// SIMATIC S7-200 project (STEP 7-Micro/WIN), CPU 224 REL 02.01

SYMBOL_TABLE USER1
start            M0.0     // khoi dong
stopp            M0.1     // dung dong co
CBT              M0.2     // cam bien quay phai
CBP              M0.3     // cam bien quay trai
QT               M0.4     // QUAY TRAI
QP               M0.5     // QUAY PHAI
END_SYMBOL_TABLE

ORGANIZATION_BLOCK MAIN:OB1
TITLE=PROGRAM COMMENTS
BEGIN
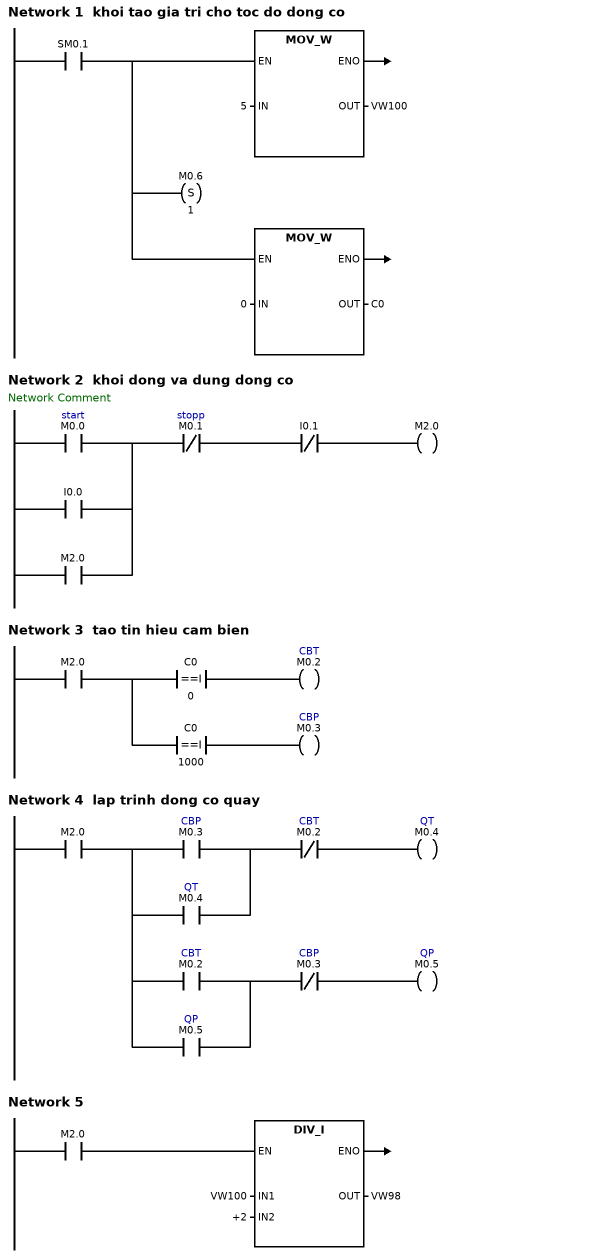
Network 1 // khoi tao gia tri cho toc do dong co
LD     SM0.1
MOVW   5, VW100
S      M0.6, 1
MOVW   0, C0
Network 2 // khoi dong va dung dong co
// Network Comment
LD     start:M0.0
O      I0.0
O      M2.0
AN     stopp:M0.1
AN     I0.1
=      M2.0
Network 3 // tao tin hieu cam bien
LD     M2.0
LPS
AW=    C0, 0
=      CBT:M0.2
LPP
AW=    C0, 1000
=      CBP:M0.3
Network 4 // lap trinh dong co quay
LD     M2.0
LPS
LD     CBP:M0.3
O      QT:M0.4
ALD
AN     CBT:M0.2
=      QT:M0.4
LPP
LD     CBT:M0.2
O      QP:M0.5
ALD
AN     CBP:M0.3
=      QP:M0.5
Network 5
LD     M2.0
MOVW   VW100, VW98
/I     +2, VW98
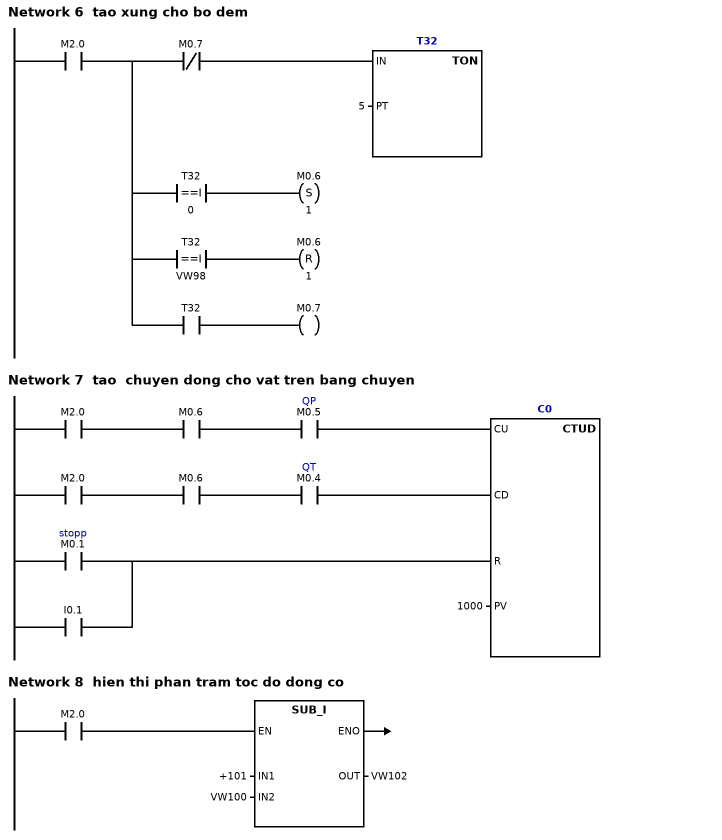
Network 6 // tao xung cho bo dem
LD     M2.0
LPS
AN     M0.7
TON    T32, 5
LRD
AW=    T32, 0
S      M0.6, 1
LRD
AW=    T32, VW98
R      M0.6, 1
LPP
A      T32
=      M0.7
Network 7 // tao  chuyen dong cho vat tren bang chuyen
LD     M2.0
A      M0.6
A      QP:M0.5
LD     M2.0
A      M0.6
A      QT:M0.4
LD     stopp:M0.1
O      I0.1
CTUD   C0, 1000
Network 8 // hien thi phan tram toc do dong co
LD     M2.0
MOVW   +101, VW102
-I     VW100, VW102
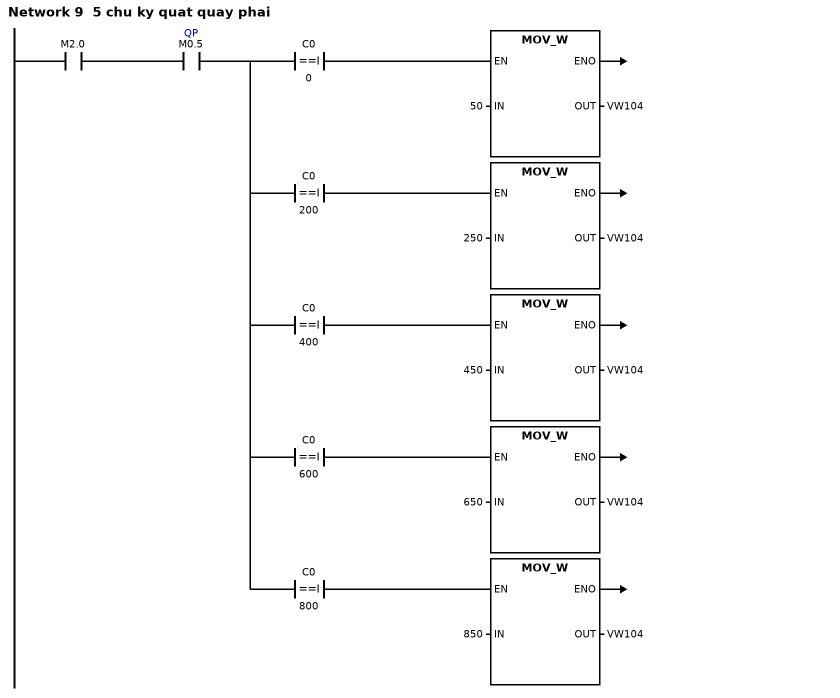
Network 9 // 5 chu ky quat quay phai
LD     M2.0
A      QP:M0.5
LPS
AW=    C0, 0
MOVW   50, VW104
LRD
AW=    C0, 200
MOVW   250, VW104
LRD
AW=    C0, 400
MOVW   450, VW104
LRD
AW=    C0, 600
MOVW   650, VW104
LPP
AW=    C0, 800
MOVW   850, VW104
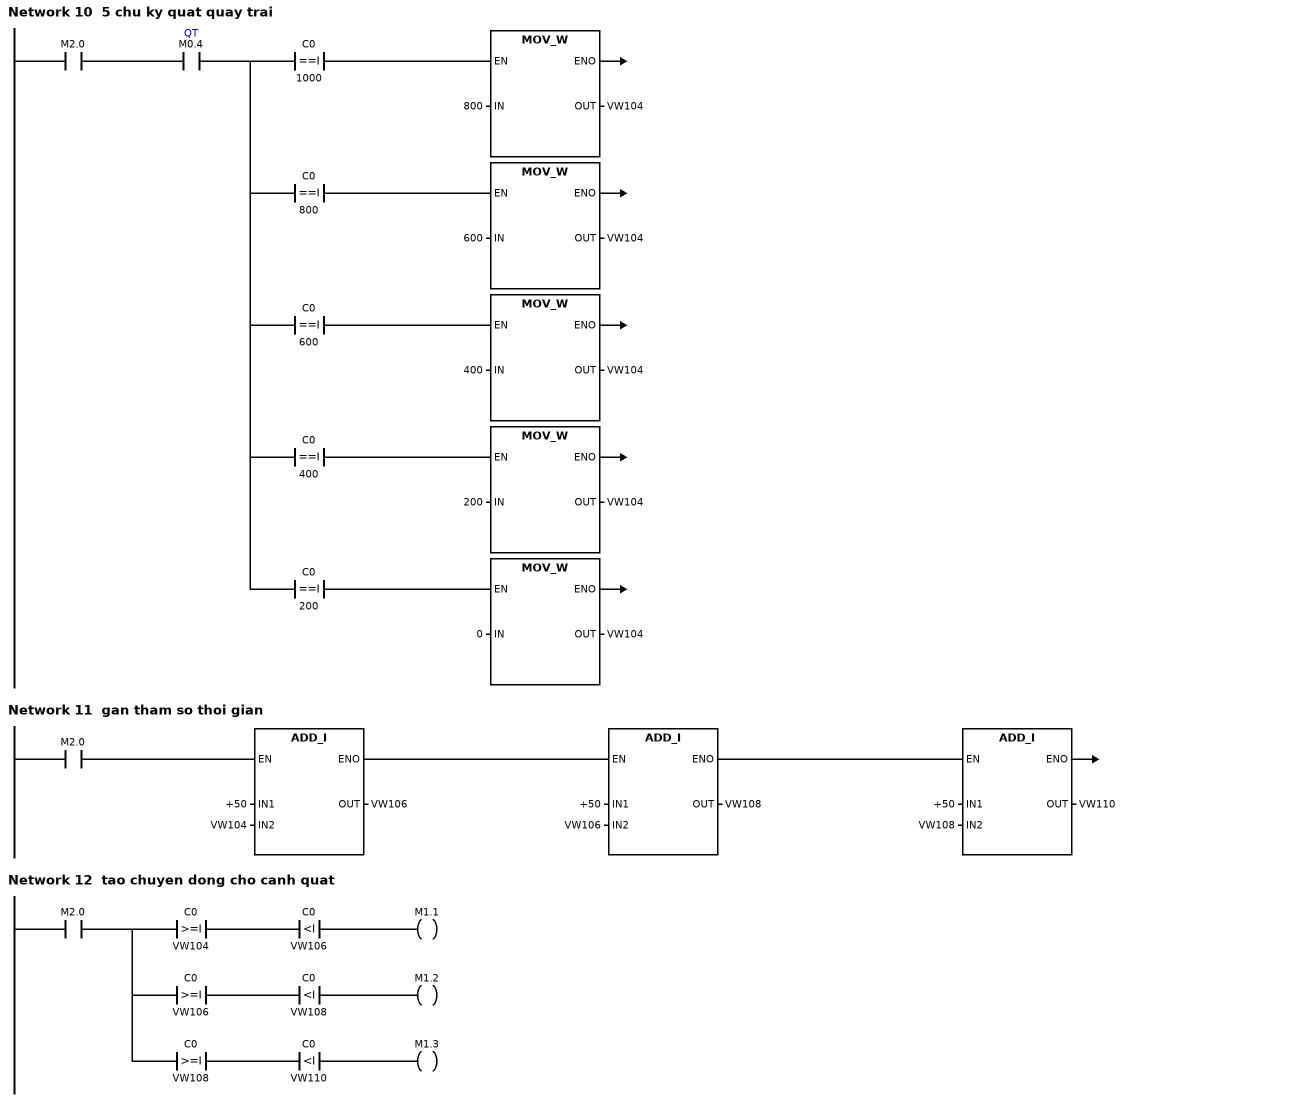
Network 10 // 5 chu ky quat quay trai
LD     M2.0
A      QT:M0.4
LPS
AW=    C0, 1000
MOVW   800, VW104
LRD
AW=    C0, 800
MOVW   600, VW104
LRD
AW=    C0, 600
MOVW   400, VW104
LRD
AW=    C0, 400
MOVW   200, VW104
LPP
AW=    C0, 200
MOVW   0, VW104
Network 11 // gan tham so thoi gian
LD     M2.0
MOVW   +50, VW106
AENO
+I     VW104, VW106
AENO
MOVW   +50, VW108
AENO
+I     VW106, VW108
AENO
MOVW   +50, VW110
+I     VW108, VW110
Network 12 // tao chuyen dong cho canh quat
LD     M2.0
LPS
AW>=   C0, VW104
AW<    C0, VW106
=      M1.1
LRD
AW>=   C0, VW106
AW<    C0, VW108
=      M1.2
LPP
AW>=   C0, VW108
AW<    C0, VW110
=      M1.3
END_ORGANIZATION_BLOCK
